
FUNCTION CB_bool_to_real : REAL


TITLE = ' Convert a boolean into a real '
VERSION : '1.0'
AUTHOR  : CB
NAME    : boToReal
FAMILY  : TNI

VAR_INPUT
    IN : BOOL;
END_VAR

VAR_TEMP

END_VAR

BEGIN

CB_bool_to_real := DINT_TO_REAL(BOOL_TO_DINT(IN));

END_FUNCTION
